(* CoDeSys 2.3.9.62 project: AperturaConClave.pro *)
(* Libraries: Standard.lib 2.6.14 11:37:46 *)

(* Global variable list: Global_Variables *)
VAR_GLOBAL

   (* Entradas *)
  (* Botonera de entrada *)
   Ent1:BOOL;
   Ent2:BOOL;
   Ent3:BOOL;
   Ent4:BOOL;
   Cierre:BOOL;



   (* Salidas *)
   CajaAbierta: BOOL;

   (*Claves *)
   Clave1:INT:=1;
  Clave2:INT:=2;
  Clave3:INT:=2;

   Valor:INT;
   Pulsacion:BOOL;
	E0:BOOL;
	E1:BOOL;
	E2:BOOL;
	E3:BOOL;
	E4:BOOL;
	Cont:INT;
END_VAR

(* POU PLC_PRG, ST *)
PROGRAM PLC_PRG
VAR
	Dig: INT;
	Salida: BOOL;
	Val: INT;
END_VAR
Val:=AutomatismoClave();
Automatismo();

IF(NOT (E0 OR E1 OR E2 OR E3)) THEN
	E0:=TRUE;
END_IF

IF(Pulsacion) THEN
	IF(E0 AND Pulsacion AND Val=Clave1) THEN
		E0:=FALSE;
		E1:=TRUE;
		Salida:=TRUE;
	ELSIF (E1 AND Pulsacion AND Val=Clave2) THEN
		E1:=FALSE;
		E2:=TRUE;
		Salida:=TRUE;
	ELSIF(E2 AND Pulsacion AND Val=Clave3) THEN
		E2:=FALSE;
		E3:=TRUE;
		Salida:=TRUE;
	ELSE
		Salida:=FALSE;
		E0:=TRUE;
		E1:=FALSE;
		E2:=FALSE;
		E3:=FALSE;
	END_IF
END_IF

IF(E3 AND Salida) THEN
	CajaAbierta:=TRUE;
END_IF

IF(E3 AND Cierre) THEN
CajaAbierta:=FALSE;
E3:=FALSE;
E0:=TRUE;
END_IF
END_PROGRAM

(* POU AutomatismoClave, ST *)
FUNCTION AutomatismoClave : INT
VAR_INPUT
END_VAR
VAR
	Val:INT;
END_VAR
IF(Ent1) THEN Val:=1; END_IF
IF(Ent2) THEN Val:=2; END_IF
IF(Ent3) THEN Val:=3; END_IF
IF(Ent4) THEN Val:=4; END_IF

AutomatismoClave:=Val;
END_FUNCTION

(* POU Automatismo, LD *)
FUNCTION Automatismo:BOOL
VAR_INPUT
END_VAR
VAR
	Contador: CTU;
	Q: BOOL;
END_VAR
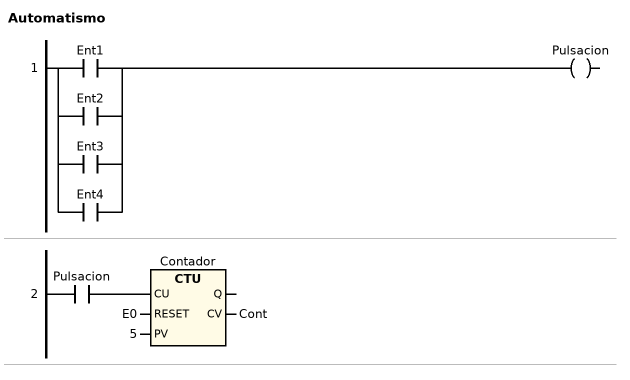
_LD_ (* Ladder Diagram *)
NETWORK 1
	{ [Ent1] | [Ent2] | [Ent3] | [Ent4] } --- (Pulsacion)
NETWORK 2
	[Pulsacion] - Contador:CTU(CU: *, RESET: E0, PV: 5, CV => Cont)
_END_LD_
(* the same logic as Structured Text *)
(* Network 1 *)
Pulsacion := Ent1 OR Ent2 OR Ent3 OR Ent4;
(* Network 2 *)
Contador(CU := Pulsacion, RESET := E0, PV := 5);
Cont := Contador.CV;
END_FUNCTION

(* Visualisation Visu
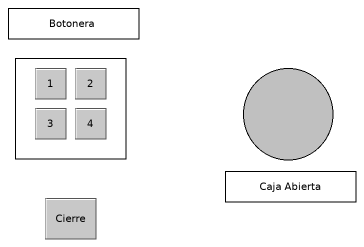
button at (50,130)-(81,161): text "1"; taps Ent1
button at (90,130)-(121,161): text "2"; taps Ent2
button at (50,170)-(81,201): text "3"; taps Ent3
button at (90,170)-(121,201): text "4"; taps Ent4
button at (60,260)-(111,301): text "Cierre"; taps Cierre
rectangle at (23,70)-(154,101): text "Botonera"
ellipse at (258,130)-(348,222): alarm colour if CajaAbierta
rectangle at (240,233)-(371,264): text "Caja Abierta"
1 more shapes without text or variables
*)
